PROGRAM PRG_Safe
VAR
	edgeDetectorBtnYellow	: Fb_EdgeDetector;
	edgeDetectorBtnBlue		: Fb_EdgeDetector;
	programmingDone			: BOOL;
	codeArray				: ARRAY [1..codeDigits] OF BOOL;
	currentIndex			: INT; 
	correctCounter			: INT; 
	timer					: TON;
	
END_VAR
VAR CONSTANT
	lightDuration			: TIME := T#5S;   // (seconds)
	codeDigits				: INT := 4;
END_VAR

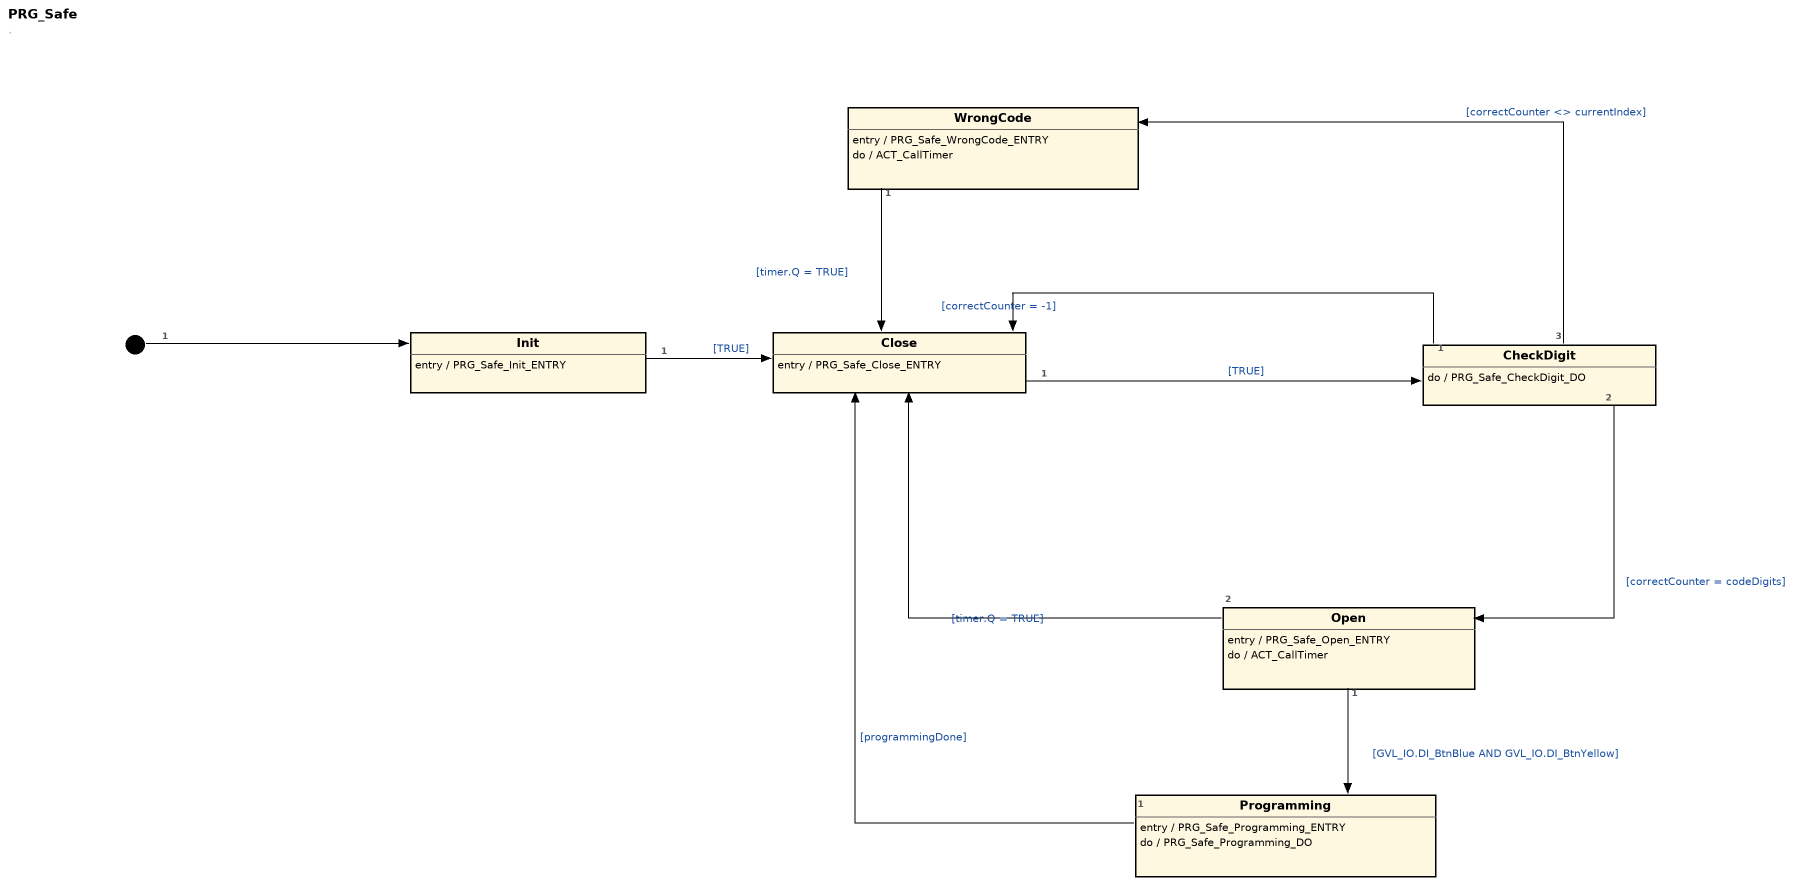
STATECHART PRG_Safe  // abortable
    START StartState1
    NOTEELEMENT 
    STATE WrongCode
        entry / PRG_Safe_WrongCode_ENTRY
        do / ACT_CallTimer
    STATE Init
        entry / PRG_Safe_Init_ENTRY
    STATE Close
        entry / PRG_Safe_Close_ENTRY
    STATE CheckDigit
        do / PRG_Safe_CheckDigit_DO
    STATE Open
        entry / PRG_Safe_Open_ENTRY
        do / ACT_CallTimer
    STATE Programming
        entry / PRG_Safe_Programming_ENTRY
        do / PRG_Safe_Programming_DO
    StartState1 -> Init  // priority 1, on completion
    WrongCode -> Close [timer.Q = TRUE] // priority 1
    Init -> Close [TRUE] // priority 1
    Close -> CheckDigit [TRUE] // priority 1
    CheckDigit -> Close [correctCounter = -1] // priority 1
    CheckDigit -> Open [correctCounter = codeDigits] // priority 2
    CheckDigit -> WrongCode [correctCounter <> currentIndex] // priority 3
    Open -> Programming [GVL_IO.DI_BtnBlue AND GVL_IO.DI_BtnYellow] // priority 1
    Open -> Close [timer.Q = TRUE] // priority 2
    Programming -> Close [programmingDone] // priority 1
END_STATECHART

ACTION ACT_CallTimer:
// call timer function block
timer();
END_ACTION

ACTION PRG_Safe_CheckDigit_DO:
// run edgedetectors
edgeDetectorBtnYellow(inputValue := GVL_IO.DI_BtnYellow);
edgeDetectorBtnBlue(inputValue := GVL_IO.DI_BtnBlue);

// any rising edges?
IF edgeDetectorBtnYellow.risingEdge OR edgeDetectorBtnBlue.risingEdge THEN
	
	// the correct button was pressed
	IF (codeArray[currentIndex+1] = TRUE   AND edgeDetectorBtnYellow.risingEdge) OR
	   (codeArray[currentIndex+1] = FALSE  AND edgeDetectorBtnBlue.risingEdge)   THEN
		correctCounter := correctCounter + 1;
		
	// the wrong button was pressed	
	ELSE
		correctCounter := 0;
	END_IF
	
	currentIndex := currentIndex + 1;
	
END_IF


// double tap blue button
IF edgeDetectorBtnBlue.doublePress THEN
	// will trigger the state change to abort code entry
	correctCounter := -1;
END_IF
END_ACTION

ACTION PRG_Safe_Close_ENTRY:
// reset outputs
GVL_IO.DO_LampGreen := FALSE;
GVL_IO.DO_LampRed := FALSE;

// reset all variables
currentIndex := 0;
correctCounter := 0;
programmingDone := FALSE;

// stop timer
timer.IN := FALSE;
timer();  // call timer so that it resets itself
END_ACTION

ACTION PRG_Safe_Init_ENTRY:
// register correct code
codeArray[1] := TRUE; 
codeArray[2] := FALSE; 
codeArray[3] := TRUE; 
codeArray[4] := FALSE;
END_ACTION

ACTION PRG_Safe_Open_ENTRY:
// light up green lamp
GVL_IO.DO_LampGreen := TRUE;

// configure and start timer
timer.PT := lightDuration;
timer.IN := TRUE;
timer();
END_ACTION

ACTION PRG_Safe_Programming_DO:
// wait until timer is done
timer();
// run edgedetectors
edgeDetectorBtnYellow(inputValue := GVL_IO.DI_BtnYellow);
edgeDetectorBtnBlue(inputValue := GVL_IO.DI_BtnBlue);

IF (timer.Q = FALSE) THEN
	RETURN;
END_IF

// TIMER DONE => proceed

// any rising edges?
IF edgeDetectorBtnYellow.risingEdge OR edgeDetectorBtnBlue.risingEdge THEN
	
	IF edgeDetectorBtnYellow.risingEdge THEN
		codeArray[currentIndex+1] := TRUE;
	ELSIF edgeDetectorBtnBlue.risingEdge THEN
		codeArray[currentIndex+1] := FALSE;
	END_IF
	
	currentIndex := currentIndex + 1;
	
	// finished programming new code
	IF currentIndex = codeDigits THEN
		programmingDone := TRUE;
	END_IF

END_IF
END_ACTION

ACTION PRG_Safe_Programming_ENTRY:
// reset current index
currentIndex := 0;

// signalized programming mode
GVL_IO.DO_LampGreen := TRUE;
GVL_IO.DO_LampRed := TRUE;
timer(IN := FALSE); // reset timer
timer.PT := T#1S;
timer(IN := TRUE); // run timer
END_ACTION

ACTION PRG_Safe_WrongCode_ENTRY:
// light up red lamp
GVL_IO.DO_LampRed := TRUE;

// configure and start timer
timer.PT := lightDuration;
timer.IN := TRUE;
timer();
END_ACTION

END_PROGRAM

(* stored: Version 1.1.0.1, ProductVersion 3.1.4024.9
   POU PRG_Safe: Id {0e27d1d1-2e71-40a6-94a3-3507cbb37083}, SpecialFunc None
   Action ACT_CallTimer: Id {7728701a-40ff-47d8-840c-b774073dfc56}
   Action PRG_Safe_CheckDigit_DO: Id {3a89dd57-44c4-43a6-8811-c76a58e0f83f}
   Action PRG_Safe_Close_ENTRY: Id {123f5087-6631-476c-90f6-5293b582edb2}
   Action PRG_Safe_Init_ENTRY: Id {e40837ab-3a6c-45d1-96e7-0261f87908e1}
   Action PRG_Safe_Open_ENTRY: Id {04052505-5018-4b14-bab2-1192caca586c}
   Action PRG_Safe_Programming_DO: Id {860780e5-6822-4873-aeb9-9931c2f9ed15}
   Action PRG_Safe_Programming_ENTRY: Id {d1f6f083-d5ff-414c-8255-951ec3a6e2da}
   Action PRG_Safe_WrongCode_ENTRY: Id {8b193f0a-919d-42b5-a747-c807ff8582a8} *)
